IF xRaport THEN
	sDane := '';
	xRaport := FALSE;
	IF intStatus <> intStatusZaraportowana THEN
		intStatusZaraportowana := intStatus;
		fnKomunikatDaneDodaj_xOverFlow(sDane := sDane , sAtrybut := 'STATUS=' , sWartosc := INT_TO_STRING(intStatus) , xOverFlow := xOverFlow);	
		IF xOverFlow = TRUE THEN
			fnZapiszKomunikat(	sCalyKomunikat := '' ,
						sTypKomunikatu := 'M' ,
						sMnemonik := sMnemonik ,
						sMACAdres := sMACAdres ,
						sIDNadawcy := sIdInstancji ,
						sIDOdbiorcy := sIdAplikacji ,
						sDaneZapasowe := sDaneZapasowe ,
						sDane := sDane ,
						arTablicaKomunikatow := arTablicaKomunikatow ,
						intTablicaKomunikatowZnacznikZapisu := intTablicaKomunikatowZnacznikZapisu ,
						intTablicaKomunikatowRozmiar := intTablicaKomunikatowRozmiar ,
						sWyslanyKomunikat := sWyslanyKomunikatDummy);
			sDane := '';
		END_IF	
	END_IF	
	//Napięcia fazowe
	IF rNapiecieL1 <> rNapiecieL1Zaraportowana THEN
		rNapiecieL1Zaraportowana := rNapiecieL1;
		fnKomunikatDaneDodaj_xOverFlow(sDane := sDane , sAtrybut := 'VOLTL1=' , sWartosc := REAL_TO_STRING(rNapiecieL1) , xOverFlow := xOverFlow);	
		IF xOverFlow = TRUE THEN
			fnZapiszKomunikat(	sCalyKomunikat := '' ,
						sTypKomunikatu := 'M' ,
						sMnemonik := sMnemonik ,
						sMACAdres := sMACAdres ,
						sIDNadawcy := sIdInstancji ,
						sIDOdbiorcy := sIdAplikacji ,
						sDaneZapasowe := sDaneZapasowe ,
						sDane := sDane ,
						arTablicaKomunikatow := arTablicaKomunikatow ,
						intTablicaKomunikatowZnacznikZapisu := intTablicaKomunikatowZnacznikZapisu ,
						intTablicaKomunikatowRozmiar := intTablicaKomunikatowRozmiar ,
						sWyslanyKomunikat := sWyslanyKomunikatDummy);
			sDane := '';
		END_IF	
	END_IF
	IF rNapiecieL2 <> rNapiecieL2Zaraportowana THEN
		rNapiecieL2Zaraportowana := rNapiecieL2;
		fnKomunikatDaneDodaj_xOverFlow(sDane := sDane , sAtrybut := 'VOLTL2=' , sWartosc := REAL_TO_STRING(rNapiecieL2) , xOverFlow := xOverFlow);	
		IF xOverFlow = TRUE THEN
			fnZapiszKomunikat(	sCalyKomunikat := '' ,
						sTypKomunikatu := 'M' ,
						sMnemonik := sMnemonik ,
						sMACAdres := sMACAdres ,
						sIDNadawcy := sIdInstancji ,
						sIDOdbiorcy := sIdAplikacji ,
						sDaneZapasowe := sDaneZapasowe ,
						sDane := sDane ,
						arTablicaKomunikatow := arTablicaKomunikatow ,
						intTablicaKomunikatowZnacznikZapisu := intTablicaKomunikatowZnacznikZapisu ,
						intTablicaKomunikatowRozmiar := intTablicaKomunikatowRozmiar ,
						sWyslanyKomunikat := sWyslanyKomunikatDummy);
			sDane := '';
		END_IF	
	END_IF	
	IF rNapiecieL3 <> rNapiecieL3Zaraportowana THEN
		rNapiecieL3Zaraportowana := rNapiecieL3;
		fnKomunikatDaneDodaj_xOverFlow(sDane := sDane , sAtrybut := 'VOLTL3=' , sWartosc := REAL_TO_STRING(rNapiecieL3) , xOverFlow := xOverFlow);
		IF xOverFlow = TRUE THEN
			fnZapiszKomunikat(	sCalyKomunikat := '' ,
						sTypKomunikatu := 'M' ,
						sMnemonik := sMnemonik ,
						sMACAdres := sMACAdres ,
						sIDNadawcy := sIdInstancji ,
						sIDOdbiorcy := sIdAplikacji ,
						sDaneZapasowe := sDaneZapasowe ,
						sDane := sDane ,
						arTablicaKomunikatow := arTablicaKomunikatow ,
						intTablicaKomunikatowZnacznikZapisu := intTablicaKomunikatowZnacznikZapisu ,
						intTablicaKomunikatowRozmiar := intTablicaKomunikatowRozmiar ,
						sWyslanyKomunikat := sWyslanyKomunikatDummy);
			sDane := '';
		END_IF		
	END_IF
	//Napięcia przewodowe		
	IF rNapiecieL1L2 <> rNapiecieL1L2Zaraportowana THEN
		rNapiecieL1L2Zaraportowana := rNapiecieL1L2;
		fnKomunikatDaneDodaj_xOverFlow(sDane := sDane , sAtrybut := 'VOLTL1L2=' , sWartosc := REAL_TO_STRING(rNapiecieL1L2) , xOverFlow := xOverFlow);	
		IF xOverFlow = TRUE THEN
			fnZapiszKomunikat(	sCalyKomunikat := '' ,
						sTypKomunikatu := 'M' ,
						sMnemonik := sMnemonik ,
						sMACAdres := sMACAdres ,
						sIDNadawcy := sIdInstancji ,
						sIDOdbiorcy := sIdAplikacji ,
						sDaneZapasowe := sDaneZapasowe ,
						sDane := sDane ,
						arTablicaKomunikatow := arTablicaKomunikatow ,
						intTablicaKomunikatowZnacznikZapisu := intTablicaKomunikatowZnacznikZapisu ,
						intTablicaKomunikatowRozmiar := intTablicaKomunikatowRozmiar ,
						sWyslanyKomunikat := sWyslanyKomunikatDummy);
			sDane := '';
		END_IF	
	END_IF
	IF rNapiecieL2L3 <> rNapiecieL2L3Zaraportowana THEN
		rNapiecieL2L3Zaraportowana := rNapiecieL2L3;
		fnKomunikatDaneDodaj_xOverFlow(sDane := sDane , sAtrybut := 'VOLTL2L3=' , sWartosc := REAL_TO_STRING(rNapiecieL2L3) , xOverFlow := xOverFlow);	
		IF xOverFlow = TRUE THEN
			fnZapiszKomunikat(	sCalyKomunikat := '' ,
						sTypKomunikatu := 'M' ,
						sMnemonik := sMnemonik ,
						sMACAdres := sMACAdres ,
						sIDNadawcy := sIdInstancji ,
						sIDOdbiorcy := sIdAplikacji ,
						sDaneZapasowe := sDaneZapasowe ,
						sDane := sDane ,
						arTablicaKomunikatow := arTablicaKomunikatow ,
						intTablicaKomunikatowZnacznikZapisu := intTablicaKomunikatowZnacznikZapisu ,
						intTablicaKomunikatowRozmiar := intTablicaKomunikatowRozmiar ,
						sWyslanyKomunikat := sWyslanyKomunikatDummy);
			sDane := '';
		END_IF	
	END_IF	
	IF rNapiecieL3L1 <> rNapiecieL3L1Zaraportowana THEN
		rNapiecieL3L1Zaraportowana := rNapiecieL3L1;
		fnKomunikatDaneDodaj_xOverFlow(sDane := sDane , sAtrybut := 'VOLTL3L1=' , sWartosc := REAL_TO_STRING(rNapiecieL3L1) , xOverFlow := xOverFlow);	
		IF xOverFlow = TRUE THEN
			fnZapiszKomunikat(	sCalyKomunikat := '' ,
						sTypKomunikatu := 'M' ,
						sMnemonik := sMnemonik ,
						sMACAdres := sMACAdres ,
						sIDNadawcy := sIdInstancji ,
						sIDOdbiorcy := sIdAplikacji ,
						sDaneZapasowe := sDaneZapasowe ,
						sDane := sDane ,
						arTablicaKomunikatow := arTablicaKomunikatow ,
						intTablicaKomunikatowZnacznikZapisu := intTablicaKomunikatowZnacznikZapisu ,
						intTablicaKomunikatowRozmiar := intTablicaKomunikatowRozmiar ,
						sWyslanyKomunikat := sWyslanyKomunikatDummy);
			sDane := '';
		END_IF	
	END_IF
	//Częstotliwość 
	IF rCzestotliwosc <> rCzestotliwoscZaraportowana THEN
		rCzestotliwoscZaraportowana := rCzestotliwosc;
		fnKomunikatDaneDodaj_xOverFlow(sDane := sDane , sAtrybut := 'CZEST=' , sWartosc := REAL_TO_STRING(rCzestotliwosc) , xOverFlow := xOverFlow);	
		IF xOverFlow = TRUE THEN
			fnZapiszKomunikat(	sCalyKomunikat := '' ,
						sTypKomunikatu := 'M' ,
						sMnemonik := sMnemonik ,
						sMACAdres := sMACAdres ,
						sIDNadawcy := sIdInstancji ,
						sIDOdbiorcy := sIdAplikacji ,
						sDaneZapasowe := sDaneZapasowe ,
						sDane := sDane ,
						arTablicaKomunikatow := arTablicaKomunikatow ,
						intTablicaKomunikatowZnacznikZapisu := intTablicaKomunikatowZnacznikZapisu ,
						intTablicaKomunikatowRozmiar := intTablicaKomunikatowRozmiar ,
						sWyslanyKomunikat := sWyslanyKomunikatDummy);
			sDane := '';
		END_IF	
	END_IF
	//Czas pracy 
	IF rCzasPracyAnalizatora <> rCzasPracyAnalizatoraZaraportowana THEN
		rCzasPracyAnalizatoraZaraportowana := rCzasPracyAnalizatora;
		fnKomunikatDaneDodaj_xOverFlow(sDane := sDane , sAtrybut := 'CZAS=' , sWartosc := REAL_TO_STRING(rCzasPracyAnalizatora) , xOverFlow := xOverFlow);	
		IF xOverFlow = TRUE THEN
			fnZapiszKomunikat(	sCalyKomunikat := '' ,
						sTypKomunikatu := 'M' ,
						sMnemonik := sMnemonik ,
						sMACAdres := sMACAdres ,
						sIDNadawcy := sIdInstancji ,
						sIDOdbiorcy := sIdAplikacji ,
						sDaneZapasowe := sDaneZapasowe ,
						sDane := sDane ,
						arTablicaKomunikatow := arTablicaKomunikatow ,
						intTablicaKomunikatowZnacznikZapisu := intTablicaKomunikatowZnacznikZapisu ,
						intTablicaKomunikatowRozmiar := intTablicaKomunikatowRozmiar ,
						sWyslanyKomunikat := sWyslanyKomunikatDummy);
			sDane := '';
		END_IF	
	END_IF
	//Prądy fazowe	
	IF rPradL1 <> rPradL1Zaraportowana THEN
		rPradL1Zaraportowana := rPradL1;
		fnKomunikatDaneDodaj_xOverFlow(sDane := sDane , sAtrybut := 'AMPERL1=' , sWartosc := REAL_TO_STRING(rPradL1) , xOverFlow := xOverFlow);	
		IF xOverFlow = TRUE THEN
			fnZapiszKomunikat(	sCalyKomunikat := '' ,
						sTypKomunikatu := 'M' ,
						sMnemonik := sMnemonik ,
						sMACAdres := sMACAdres ,
						sIDNadawcy := sIdInstancji ,
						sIDOdbiorcy := sIdAplikacji ,
						sDaneZapasowe := sDaneZapasowe ,
						sDane := sDane ,
						arTablicaKomunikatow := arTablicaKomunikatow ,
						intTablicaKomunikatowZnacznikZapisu := intTablicaKomunikatowZnacznikZapisu ,
						intTablicaKomunikatowRozmiar := intTablicaKomunikatowRozmiar ,
						sWyslanyKomunikat := sWyslanyKomunikatDummy);
			sDane := '';
		END_IF	
	END_IF
	IF rPradL2 <> rPradL2Zaraportowana THEN
		rPradL2Zaraportowana := rPradL2;
		fnKomunikatDaneDodaj_xOverFlow(sDane := sDane , sAtrybut := 'AMPERL2=' , sWartosc := REAL_TO_STRING(rPradL2) , xOverFlow := xOverFlow);	
		IF xOverFlow = TRUE THEN
			fnZapiszKomunikat(	sCalyKomunikat := '' ,
						sTypKomunikatu := 'M' ,
						sMnemonik := sMnemonik ,
						sMACAdres := sMACAdres ,
						sIDNadawcy := sIdInstancji ,
						sIDOdbiorcy := sIdAplikacji ,
						sDaneZapasowe := sDaneZapasowe ,
						sDane := sDane ,
						arTablicaKomunikatow := arTablicaKomunikatow ,
						intTablicaKomunikatowZnacznikZapisu := intTablicaKomunikatowZnacznikZapisu ,
						intTablicaKomunikatowRozmiar := intTablicaKomunikatowRozmiar ,
						sWyslanyKomunikat := sWyslanyKomunikatDummy);
			sDane := '';
		END_IF	
	END_IF	
	IF rPradL3 <> rPradL3Zaraportowana THEN
		rPradL3Zaraportowana := rPradL3;
		fnKomunikatDaneDodaj_xOverFlow(sDane := sDane , sAtrybut := 'AMPERL3=' , sWartosc := REAL_TO_STRING(rPradL3) , xOverFlow := xOverFlow);	
		IF xOverFlow = TRUE THEN
			fnZapiszKomunikat(	sCalyKomunikat := '' ,
						sTypKomunikatu := 'M' ,
						sMnemonik := sMnemonik ,
						sMACAdres := sMACAdres ,
						sIDNadawcy := sIdInstancji ,
						sIDOdbiorcy := sIdAplikacji ,
						sDaneZapasowe := sDaneZapasowe ,
						sDane := sDane ,
						arTablicaKomunikatow := arTablicaKomunikatow ,
						intTablicaKomunikatowZnacznikZapisu := intTablicaKomunikatowZnacznikZapisu ,
						intTablicaKomunikatowRozmiar := intTablicaKomunikatowRozmiar ,
						sWyslanyKomunikat := sWyslanyKomunikatDummy);
			sDane := '';
		END_IF	
	END_IF
	IF rPradN <> rPradNZaraportowana THEN
		rPradNZaraportowana := rPradN;
		fnKomunikatDaneDodaj_xOverFlow(sDane := sDane , sAtrybut := 'AMPERN=' , sWartosc := REAL_TO_STRING(rPradN) , xOverFlow := xOverFlow);	
		IF xOverFlow = TRUE THEN
			fnZapiszKomunikat(	sCalyKomunikat := '' ,
						sTypKomunikatu := 'M' ,
						sMnemonik := sMnemonik ,
						sMACAdres := sMACAdres ,
						sIDNadawcy := sIdInstancji ,
						sIDOdbiorcy := sIdAplikacji ,
						sDaneZapasowe := sDaneZapasowe ,
						sDane := sDane ,
						arTablicaKomunikatow := arTablicaKomunikatow ,
						intTablicaKomunikatowZnacznikZapisu := intTablicaKomunikatowZnacznikZapisu ,
						intTablicaKomunikatowRozmiar := intTablicaKomunikatowRozmiar ,
						sWyslanyKomunikat := sWyslanyKomunikatDummy);
			sDane := '';
		END_IF	
	END_IF
	//Prądy średnie fazowe
	IF rPradSredniL1 <> rPradSredniL1Zaraportowana THEN
		rPradSredniL1Zaraportowana := rPradSredniL1;
		fnKomunikatDaneDodaj_xOverFlow(sDane := sDane , sAtrybut := 'AMPERAVGL1=' , sWartosc := REAL_TO_STRING(rPradSredniL1) , xOverFlow := xOverFlow);	
		IF xOverFlow = TRUE THEN
			fnZapiszKomunikat(	sCalyKomunikat := '' ,
						sTypKomunikatu := 'M' ,
						sMnemonik := sMnemonik ,
						sMACAdres := sMACAdres ,
						sIDNadawcy := sIdInstancji ,
						sIDOdbiorcy := sIdAplikacji ,
						sDaneZapasowe := sDaneZapasowe ,
						sDane := sDane ,
						arTablicaKomunikatow := arTablicaKomunikatow ,
						intTablicaKomunikatowZnacznikZapisu := intTablicaKomunikatowZnacznikZapisu ,
						intTablicaKomunikatowRozmiar := intTablicaKomunikatowRozmiar ,
						sWyslanyKomunikat := sWyslanyKomunikatDummy);
			sDane := '';
		END_IF	
	END_IF
	IF rPradSredniL2 <> rPradSredniL2Zaraportowana THEN
		rPradSredniL2Zaraportowana := rPradSredniL2;
		fnKomunikatDaneDodaj_xOverFlow(sDane := sDane , sAtrybut := 'AMPERAVGL2=' , sWartosc := REAL_TO_STRING(rPradSredniL2) , xOverFlow := xOverFlow);	
		IF xOverFlow = TRUE THEN
			fnZapiszKomunikat(	sCalyKomunikat := '' ,
						sTypKomunikatu := 'M' ,
						sMnemonik := sMnemonik ,
						sMACAdres := sMACAdres ,
						sIDNadawcy := sIdInstancji ,
						sIDOdbiorcy := sIdAplikacji ,
						sDaneZapasowe := sDaneZapasowe ,
						sDane := sDane ,
						arTablicaKomunikatow := arTablicaKomunikatow ,
						intTablicaKomunikatowZnacznikZapisu := intTablicaKomunikatowZnacznikZapisu ,
						intTablicaKomunikatowRozmiar := intTablicaKomunikatowRozmiar ,
						sWyslanyKomunikat := sWyslanyKomunikatDummy);
			sDane := '';
		END_IF	
	END_IF	
	IF rPradSredniL3 <> rPradSredniL3Zaraportowana THEN
		rPradSredniL3Zaraportowana := rPradSredniL3;
		fnKomunikatDaneDodaj_xOverFlow(sDane := sDane , sAtrybut := 'AMPERAVGL3=' , sWartosc := REAL_TO_STRING(rPradSredniL3) , xOverFlow := xOverFlow);
		IF xOverFlow = TRUE THEN
			fnZapiszKomunikat(	sCalyKomunikat := '' ,
						sTypKomunikatu := 'M' ,
						sMnemonik := sMnemonik ,
						sMACAdres := sMACAdres ,
						sIDNadawcy := sIdInstancji ,
						sIDOdbiorcy := sIdAplikacji ,
						sDaneZapasowe := sDaneZapasowe ,
						sDane := sDane ,
						arTablicaKomunikatow := arTablicaKomunikatow ,
						intTablicaKomunikatowZnacznikZapisu := intTablicaKomunikatowZnacznikZapisu ,
						intTablicaKomunikatowRozmiar := intTablicaKomunikatowRozmiar ,
						sWyslanyKomunikat := sWyslanyKomunikatDummy);
			sDane := '';
		END_IF	
	END_IF
	//Prąd średni
	IF rPradSredni <> rPradSredniZaraportowana THEN
		rPradSredniZaraportowana := rPradSredni;
		fnKomunikatDaneDodaj_xOverFlow(sDane := sDane , sAtrybut := 'AMPERAVG=' , sWartosc := REAL_TO_STRING(rPradSredni) , xOverFlow := xOverFlow);
		IF xOverFlow = TRUE THEN
			fnZapiszKomunikat(	sCalyKomunikat := '' ,
						sTypKomunikatu := 'M' ,
						sMnemonik := sMnemonik ,
						sMACAdres := sMACAdres ,
						sIDNadawcy := sIdInstancji ,
						sIDOdbiorcy := sIdAplikacji ,
						sDaneZapasowe := sDaneZapasowe ,
						sDane := sDane ,
						arTablicaKomunikatow := arTablicaKomunikatow ,
						intTablicaKomunikatowZnacznikZapisu := intTablicaKomunikatowZnacznikZapisu ,
						intTablicaKomunikatowRozmiar := intTablicaKomunikatowRozmiar ,
						sWyslanyKomunikat := sWyslanyKomunikatDummy);
			sDane := '';
		END_IF	
	END_IF
	//Moce 3-fazowe		 
	IF rMocCzynnaCalkowita <> rMocCzynnaCalkowitaZaraportowana THEN
		rMocCzynnaCalkowitaZaraportowana := rMocCzynnaCalkowita;
		fnKomunikatDaneDodaj_xOverFlow(sDane := sDane , sAtrybut := 'POWCE=' , sWartosc := REAL_TO_STRING(rMocCzynnaCalkowita) , xOverFlow := xOverFlow);
		IF xOverFlow = TRUE THEN
			fnZapiszKomunikat(	sCalyKomunikat := '' ,
						sTypKomunikatu := 'M' ,
						sMnemonik := sMnemonik ,
						sMACAdres := sMACAdres ,
						sIDNadawcy := sIdInstancji ,
						sIDOdbiorcy := sIdAplikacji ,
						sDaneZapasowe := sDaneZapasowe ,
						sDane := sDane ,
						arTablicaKomunikatow := arTablicaKomunikatow ,
						intTablicaKomunikatowZnacznikZapisu := intTablicaKomunikatowZnacznikZapisu ,
						intTablicaKomunikatowRozmiar := intTablicaKomunikatowRozmiar ,
						sWyslanyKomunikat := sWyslanyKomunikatDummy);
			sDane := '';
		END_IF	
	END_IF
	IF rMocBiernaCalkowita <> rMocBiernaCalkowitaZaraportowana THEN
		rMocBiernaCalkowitaZaraportowana := rMocBiernaCalkowita;
		fnKomunikatDaneDodaj_xOverFlow(sDane := sDane , sAtrybut := 'POWBE=' , sWartosc := REAL_TO_STRING(rMocBiernaCalkowita) , xOverFlow := xOverFlow);	
		IF xOverFlow = TRUE THEN
			fnZapiszKomunikat(	sCalyKomunikat := '' ,
						sTypKomunikatu := 'M' ,
						sMnemonik := sMnemonik ,
						sMACAdres := sMACAdres ,
						sIDNadawcy := sIdInstancji ,
						sIDOdbiorcy := sIdAplikacji ,
						sDaneZapasowe := sDaneZapasowe ,
						sDane := sDane ,
						arTablicaKomunikatow := arTablicaKomunikatow ,
						intTablicaKomunikatowZnacznikZapisu := intTablicaKomunikatowZnacznikZapisu ,
						intTablicaKomunikatowRozmiar := intTablicaKomunikatowRozmiar ,
						sWyslanyKomunikat := sWyslanyKomunikatDummy);
			sDane := '';
		END_IF	
	END_IF	
	IF rMocPozornaCalkowita <> rMocPozornaCalkowitaZaraportowana THEN
		rMocPozornaCalkowitaZaraportowana := rMocPozornaCalkowita;
		fnKomunikatDaneDodaj_xOverFlow(sDane := sDane , sAtrybut := 'POWPE=' , sWartosc := REAL_TO_STRING(rMocPozornaCalkowita) , xOverFlow := xOverFlow);	
		IF xOverFlow = TRUE THEN
			fnZapiszKomunikat(	sCalyKomunikat := '' ,
						sTypKomunikatu := 'M' ,
						sMnemonik := sMnemonik ,
						sMACAdres := sMACAdres ,
						sIDNadawcy := sIdInstancji ,
						sIDOdbiorcy := sIdAplikacji ,
						sDaneZapasowe := sDaneZapasowe ,
						sDane := sDane ,
						arTablicaKomunikatow := arTablicaKomunikatow ,
						intTablicaKomunikatowZnacznikZapisu := intTablicaKomunikatowZnacznikZapisu ,
						intTablicaKomunikatowRozmiar := intTablicaKomunikatowRozmiar ,
						sWyslanyKomunikat := sWyslanyKomunikatDummy);
			sDane := '';
		END_IF	
	END_IF
	//Współczynnik mocy 3-fazowy
	IF rWspolczynnikMocyCalkowity <> rWspolczynnikMocyCalkowityZaraportowana THEN
		rWspolczynnikMocyCalkowityZaraportowana := rWspolczynnikMocyCalkowity;
		fnKomunikatDaneDodaj_xOverFlow(sDane := sDane , sAtrybut := 'FACTOR3PH=' , sWartosc := REAL_TO_STRING(rWspolczynnikMocyCalkowity) , xOverFlow := xOverFlow);	
		IF xOverFlow = TRUE THEN
			fnZapiszKomunikat(	sCalyKomunikat := '' ,
						sTypKomunikatu := 'M' ,
						sMnemonik := sMnemonik ,
						sMACAdres := sMACAdres ,
						sIDNadawcy := sIdInstancji ,
						sIDOdbiorcy := sIdAplikacji ,
						sDaneZapasowe := sDaneZapasowe ,
						sDane := sDane ,
						arTablicaKomunikatow := arTablicaKomunikatow ,
						intTablicaKomunikatowZnacznikZapisu := intTablicaKomunikatowZnacznikZapisu ,
						intTablicaKomunikatowRozmiar := intTablicaKomunikatowRozmiar ,
						sWyslanyKomunikat := sWyslanyKomunikatDummy);
			sDane := '';
		END_IF	
	END_IF
	//Moce czynne fazowe
	IF rMocCzynnaL1 <> rMocCzynnaL1Zaraportowana THEN
		rMocCzynnaL1Zaraportowana := rMocCzynnaL1;
		fnKomunikatDaneDodaj_xOverFlow(sDane := sDane , sAtrybut := 'POWCECL1=' , sWartosc := REAL_TO_STRING(rMocCzynnaL1) , xOverFlow := xOverFlow);	
		IF xOverFlow = TRUE THEN
			fnZapiszKomunikat(	sCalyKomunikat := '' ,
						sTypKomunikatu := 'M' ,
						sMnemonik := sMnemonik ,
						sMACAdres := sMACAdres ,
						sIDNadawcy := sIdInstancji ,
						sIDOdbiorcy := sIdAplikacji ,
						sDaneZapasowe := sDaneZapasowe ,
						sDane := sDane ,
						arTablicaKomunikatow := arTablicaKomunikatow ,
						intTablicaKomunikatowZnacznikZapisu := intTablicaKomunikatowZnacznikZapisu ,
						intTablicaKomunikatowRozmiar := intTablicaKomunikatowRozmiar ,
						sWyslanyKomunikat := sWyslanyKomunikatDummy);
			sDane := '';
		END_IF	
	END_IF
	IF rMocCzynnaL2 <> rMocCzynnaL2Zaraportowana THEN
		rMocCzynnaL2Zaraportowana := rMocCzynnaL2;
		fnKomunikatDaneDodaj_xOverFlow(sDane := sDane , sAtrybut := 'POWCECL2=' , sWartosc := REAL_TO_STRING(rMocCzynnaL2) , xOverFlow := xOverFlow);	
		IF xOverFlow = TRUE THEN
			fnZapiszKomunikat(	sCalyKomunikat := '' ,
						sTypKomunikatu := 'M' ,
						sMnemonik := sMnemonik ,
						sMACAdres := sMACAdres ,
						sIDNadawcy := sIdInstancji ,
						sIDOdbiorcy := sIdAplikacji ,
						sDaneZapasowe := sDaneZapasowe ,
						sDane := sDane ,
						arTablicaKomunikatow := arTablicaKomunikatow ,
						intTablicaKomunikatowZnacznikZapisu := intTablicaKomunikatowZnacznikZapisu ,
						intTablicaKomunikatowRozmiar := intTablicaKomunikatowRozmiar ,
						sWyslanyKomunikat := sWyslanyKomunikatDummy);
			sDane := '';
		END_IF	
	END_IF
	IF rMocCzynnaL3 <> rMocCzynnaL3Zaraportowana THEN
		rMocCzynnaL3Zaraportowana := rMocCzynnaL3;
		fnKomunikatDaneDodaj_xOverFlow(sDane := sDane , sAtrybut := 'POWCECL3=' , sWartosc := REAL_TO_STRING(rMocCzynnaL3) , xOverFlow := xOverFlow);
		IF xOverFlow = TRUE THEN
			fnZapiszKomunikat(	sCalyKomunikat := '' ,
						sTypKomunikatu := 'M' ,
						sMnemonik := sMnemonik ,
						sMACAdres := sMACAdres ,
						sIDNadawcy := sIdInstancji ,
						sIDOdbiorcy := sIdAplikacji ,
						sDaneZapasowe := sDaneZapasowe ,
						sDane := sDane ,
						arTablicaKomunikatow := arTablicaKomunikatow ,
						intTablicaKomunikatowZnacznikZapisu := intTablicaKomunikatowZnacznikZapisu ,
						intTablicaKomunikatowRozmiar := intTablicaKomunikatowRozmiar ,
						sWyslanyKomunikat := sWyslanyKomunikatDummy);
			sDane := '';
		END_IF		
	END_IF
	//Moce bierne fazowe	
	IF rMocBiernaL1 <> rMocBiernaL1Zaraportowana THEN
		rMocBiernaL1Zaraportowana := rMocBiernaL1;
		fnKomunikatDaneDodaj_xOverFlow(sDane := sDane , sAtrybut := 'POWCEBL1=' , sWartosc := REAL_TO_STRING(rMocBiernaL1) , xOverFlow := xOverFlow);	
		IF xOverFlow = TRUE THEN
			fnZapiszKomunikat(	sCalyKomunikat := '' ,
						sTypKomunikatu := 'M' ,
						sMnemonik := sMnemonik ,
						sMACAdres := sMACAdres ,
						sIDNadawcy := sIdInstancji ,
						sIDOdbiorcy := sIdAplikacji ,
						sDaneZapasowe := sDaneZapasowe ,
						sDane := sDane ,
						arTablicaKomunikatow := arTablicaKomunikatow ,
						intTablicaKomunikatowZnacznikZapisu := intTablicaKomunikatowZnacznikZapisu ,
						intTablicaKomunikatowRozmiar := intTablicaKomunikatowRozmiar ,
						sWyslanyKomunikat := sWyslanyKomunikatDummy);
			sDane := '';
		END_IF	
	END_IF
	IF rMocBiernaL2 <> rMocBiernaL2Zaraportowana THEN
		rMocBiernaL2Zaraportowana := rMocBiernaL2;
		fnKomunikatDaneDodaj_xOverFlow(sDane := sDane , sAtrybut := 'POWCEBL2=' , sWartosc := REAL_TO_STRING(rMocBiernaL2) , xOverFlow := xOverFlow);	
		IF xOverFlow = TRUE THEN
			fnZapiszKomunikat(	sCalyKomunikat := '' ,
						sTypKomunikatu := 'M' ,
						sMnemonik := sMnemonik ,
						sMACAdres := sMACAdres ,
						sIDNadawcy := sIdInstancji ,
						sIDOdbiorcy := sIdAplikacji ,
						sDaneZapasowe := sDaneZapasowe ,
						sDane := sDane ,
						arTablicaKomunikatow := arTablicaKomunikatow ,
						intTablicaKomunikatowZnacznikZapisu := intTablicaKomunikatowZnacznikZapisu ,
						intTablicaKomunikatowRozmiar := intTablicaKomunikatowRozmiar ,
						sWyslanyKomunikat := sWyslanyKomunikatDummy);
			sDane := '';
		END_IF	
	END_IF
	IF rMocBiernaL3 <> rMocBiernaL3Zaraportowana THEN
		rMocBiernaL3Zaraportowana := rMocBiernaL3;
		fnKomunikatDaneDodaj_xOverFlow(sDane := sDane , sAtrybut := 'POWCEBL3=' , sWartosc := REAL_TO_STRING(rMocBiernaL3) , xOverFlow := xOverFlow);	
		IF xOverFlow = TRUE THEN
			fnZapiszKomunikat(	sCalyKomunikat := '' ,
						sTypKomunikatu := 'M' ,
						sMnemonik := sMnemonik ,
						sMACAdres := sMACAdres ,
						sIDNadawcy := sIdInstancji ,
						sIDOdbiorcy := sIdAplikacji ,
						sDaneZapasowe := sDaneZapasowe ,
						sDane := sDane ,
						arTablicaKomunikatow := arTablicaKomunikatow ,
						intTablicaKomunikatowZnacznikZapisu := intTablicaKomunikatowZnacznikZapisu ,
						intTablicaKomunikatowRozmiar := intTablicaKomunikatowRozmiar ,
						sWyslanyKomunikat := sWyslanyKomunikatDummy);
			sDane := '';
		END_IF	
	END_IF
	//Moce pozorne fazowe
	IF rMocPozornaL1 <> rMocPozornaL1Zaraportowana THEN
		rMocPozornaL1Zaraportowana := rMocPozornaL1;
		fnKomunikatDaneDodaj_xOverFlow(sDane := sDane , sAtrybut := 'POWCEPL1=' , sWartosc := REAL_TO_STRING(rMocPozornaL1) , xOverFlow := xOverFlow);	
		IF xOverFlow = TRUE THEN
			fnZapiszKomunikat(	sCalyKomunikat := '' ,
						sTypKomunikatu := 'M' ,
						sMnemonik := sMnemonik ,
						sMACAdres := sMACAdres ,
						sIDNadawcy := sIdInstancji ,
						sIDOdbiorcy := sIdAplikacji ,
						sDaneZapasowe := sDaneZapasowe ,
						sDane := sDane ,
						arTablicaKomunikatow := arTablicaKomunikatow ,
						intTablicaKomunikatowZnacznikZapisu := intTablicaKomunikatowZnacznikZapisu ,
						intTablicaKomunikatowRozmiar := intTablicaKomunikatowRozmiar ,
						sWyslanyKomunikat := sWyslanyKomunikatDummy);
			sDane := '';
		END_IF	
	END_IF
	IF rMocPozornaL2 <> rMocPozornaL2Zaraportowana THEN
		rMocPozornaL2Zaraportowana := rMocPozornaL2;
		fnKomunikatDaneDodaj_xOverFlow(sDane := sDane , sAtrybut := 'POWCEPL2=' , sWartosc := REAL_TO_STRING(rMocPozornaL2) , xOverFlow := xOverFlow);	
		IF xOverFlow = TRUE THEN
			fnZapiszKomunikat(	sCalyKomunikat := '' ,
						sTypKomunikatu := 'M' ,
						sMnemonik := sMnemonik ,
						sMACAdres := sMACAdres ,
						sIDNadawcy := sIdInstancji ,
						sIDOdbiorcy := sIdAplikacji ,
						sDaneZapasowe := sDaneZapasowe ,
						sDane := sDane ,
						arTablicaKomunikatow := arTablicaKomunikatow ,
						intTablicaKomunikatowZnacznikZapisu := intTablicaKomunikatowZnacznikZapisu ,
						intTablicaKomunikatowRozmiar := intTablicaKomunikatowRozmiar ,
						sWyslanyKomunikat := sWyslanyKomunikatDummy);
			sDane := '';
		END_IF	
	END_IF
	IF rMocPozornaL3 <> rMocPozornaL3Zaraportowana THEN
		rMocPozornaL3Zaraportowana := rMocPozornaL3;
		fnKomunikatDaneDodaj_xOverFlow(sDane := sDane , sAtrybut := 'POWCEPL3=' , sWartosc := REAL_TO_STRING(rMocPozornaL3) , xOverFlow := xOverFlow);	
		IF xOverFlow = TRUE THEN
			fnZapiszKomunikat(	sCalyKomunikat := '' ,
						sTypKomunikatu := 'M' ,
						sMnemonik := sMnemonik ,
						sMACAdres := sMACAdres ,
						sIDNadawcy := sIdInstancji ,
						sIDOdbiorcy := sIdAplikacji ,
						sDaneZapasowe := sDaneZapasowe ,
						sDane := sDane ,
						arTablicaKomunikatow := arTablicaKomunikatow ,
						intTablicaKomunikatowZnacznikZapisu := intTablicaKomunikatowZnacznikZapisu ,
						intTablicaKomunikatowRozmiar := intTablicaKomunikatowRozmiar ,
						sWyslanyKomunikat := sWyslanyKomunikatDummy);
			sDane := '';
		END_IF	
	END_IF
	//Współczynniki mocy fazowe
	IF rWspolczynnikMocyL1 <> rWspolczynnikMocyL1Zaraportowana THEN
		rWspolczynnikMocyL1Zaraportowana := rWspolczynnikMocyL1;
		fnKomunikatDaneDodaj_xOverFlow(sDane := sDane , sAtrybut := 'FACTORL1=' , sWartosc := REAL_TO_STRING(rWspolczynnikMocyL1) , xOverFlow := xOverFlow);
		IF xOverFlow = TRUE THEN
			fnZapiszKomunikat(	sCalyKomunikat := '' ,
						sTypKomunikatu := 'M' ,
						sMnemonik := sMnemonik ,
						sMACAdres := sMACAdres ,
						sIDNadawcy := sIdInstancji ,
						sIDOdbiorcy := sIdAplikacji ,
						sDaneZapasowe := sDaneZapasowe ,
						sDane := sDane ,
						arTablicaKomunikatow := arTablicaKomunikatow ,
						intTablicaKomunikatowZnacznikZapisu := intTablicaKomunikatowZnacznikZapisu ,
						intTablicaKomunikatowRozmiar := intTablicaKomunikatowRozmiar ,
						sWyslanyKomunikat := sWyslanyKomunikatDummy);
			sDane := '';
		END_IF		
	END_IF
	IF rWspolczynnikMocyL2 <> rWspolczynnikMocyL2Zaraportowana THEN
		rWspolczynnikMocyL2Zaraportowana := rWspolczynnikMocyL2;
		fnKomunikatDaneDodaj_xOverFlow(sDane := sDane , sAtrybut := 'FACTORL2=' , sWartosc := REAL_TO_STRING(rWspolczynnikMocyL2) , xOverFlow := xOverFlow);	
		IF xOverFlow = TRUE THEN
			fnZapiszKomunikat(	sCalyKomunikat := '' ,
						sTypKomunikatu := 'M' ,
						sMnemonik := sMnemonik ,
						sMACAdres := sMACAdres ,
						sIDNadawcy := sIdInstancji ,
						sIDOdbiorcy := sIdAplikacji ,
						sDaneZapasowe := sDaneZapasowe ,
						sDane := sDane ,
						arTablicaKomunikatow := arTablicaKomunikatow ,
						intTablicaKomunikatowZnacznikZapisu := intTablicaKomunikatowZnacznikZapisu ,
						intTablicaKomunikatowRozmiar := intTablicaKomunikatowRozmiar ,
						sWyslanyKomunikat := sWyslanyKomunikatDummy);
			sDane := '';
		END_IF	
	END_IF
	IF rWspolczynnikMocyL3 <> rWspolczynnikMocyL3Zaraportowana THEN
		rWspolczynnikMocyL3Zaraportowana := rWspolczynnikMocyL3;
		fnKomunikatDaneDodaj_xOverFlow(sDane := sDane , sAtrybut := 'FACTORL3=' , sWartosc := REAL_TO_STRING(rWspolczynnikMocyL3) , xOverFlow := xOverFlow);	
		IF xOverFlow = TRUE THEN
			fnZapiszKomunikat(	sCalyKomunikat := '' ,
						sTypKomunikatu := 'M' ,
						sMnemonik := sMnemonik ,
						sMACAdres := sMACAdres ,
						sIDNadawcy := sIdInstancji ,
						sIDOdbiorcy := sIdAplikacji ,
						sDaneZapasowe := sDaneZapasowe ,
						sDane := sDane ,
						arTablicaKomunikatow := arTablicaKomunikatow ,
						intTablicaKomunikatowZnacznikZapisu := intTablicaKomunikatowZnacznikZapisu ,
						intTablicaKomunikatowRozmiar := intTablicaKomunikatowRozmiar ,
						sWyslanyKomunikat := sWyslanyKomunikatDummy);
			sDane := '';
		END_IF	
	END_IF
	//Energia pobrana
	IF rEnergiaCzynnaPobrana <> rEnergiaCzynnaPobranaZaraportowana THEN
		rEnergiaCzynnaPobranaZaraportowana := rEnergiaCzynnaPobrana;
		fnKomunikatDaneDodaj_xOverFlow(sDane := sDane , sAtrybut := 'ENCE=' , sWartosc := REAL_TO_STRING(rEnergiaCzynnaPobrana) , xOverFlow := xOverFlow);	
		IF xOverFlow = TRUE THEN
			fnZapiszKomunikat(	sCalyKomunikat := '' ,
						sTypKomunikatu := 'M' ,
						sMnemonik := sMnemonik ,
						sMACAdres := sMACAdres ,
						sIDNadawcy := sIdInstancji ,
						sIDOdbiorcy := sIdAplikacji ,
						sDaneZapasowe := sDaneZapasowe ,
						sDane := sDane ,
						arTablicaKomunikatow := arTablicaKomunikatow ,
						intTablicaKomunikatowZnacznikZapisu := intTablicaKomunikatowZnacznikZapisu ,
						intTablicaKomunikatowRozmiar := intTablicaKomunikatowRozmiar ,
						sWyslanyKomunikat := sWyslanyKomunikatDummy);
			sDane := '';
		END_IF	
	END_IF
	IF rEnergiaBiernaPobrana <> rEnergiaBiernaPobranaZaraportowana THEN
		rEnergiaBiernaPobranaZaraportowana := rEnergiaBiernaPobrana;
		fnKomunikatDaneDodaj_xOverFlow(sDane := sDane , sAtrybut := 'ENBE=' , sWartosc := REAL_TO_STRING(rEnergiaBiernaPobrana) , xOverFlow := xOverFlow);	
		IF xOverFlow = TRUE THEN
			fnZapiszKomunikat(	sCalyKomunikat := '' ,
						sTypKomunikatu := 'M' ,
						sMnemonik := sMnemonik ,
						sMACAdres := sMACAdres ,
						sIDNadawcy := sIdInstancji ,
						sIDOdbiorcy := sIdAplikacji ,
						sDaneZapasowe := sDaneZapasowe ,
						sDane := sDane ,
						arTablicaKomunikatow := arTablicaKomunikatow ,
						intTablicaKomunikatowZnacznikZapisu := intTablicaKomunikatowZnacznikZapisu ,
						intTablicaKomunikatowRozmiar := intTablicaKomunikatowRozmiar ,
						sWyslanyKomunikat := sWyslanyKomunikatDummy);
			sDane := '';
		END_IF	
	END_IF
	IF rEnergiaPozornaPobrana <> rEnergiaPozornaPobranaZaraportowana THEN
		rEnergiaPozornaPobranaZaraportowana := rEnergiaPozornaPobrana;
		fnKomunikatDaneDodaj_xOverFlow(sDane := sDane , sAtrybut := 'ENPE=' , sWartosc := REAL_TO_STRING(rEnergiaPozornaPobrana) , xOverFlow := xOverFlow);	
		IF xOverFlow = TRUE THEN
			fnZapiszKomunikat(	sCalyKomunikat := '' ,
						sTypKomunikatu := 'M' ,
						sMnemonik := sMnemonik ,
						sMACAdres := sMACAdres ,
						sIDNadawcy := sIdInstancji ,
						sIDOdbiorcy := sIdAplikacji ,
						sDaneZapasowe := sDaneZapasowe ,
						sDane := sDane ,
						arTablicaKomunikatow := arTablicaKomunikatow ,
						intTablicaKomunikatowZnacznikZapisu := intTablicaKomunikatowZnacznikZapisu ,
						intTablicaKomunikatowRozmiar := intTablicaKomunikatowRozmiar ,
						sWyslanyKomunikat := sWyslanyKomunikatDummy);
			sDane := '';
		END_IF	
	END_IF
	//Moce średnie	
	IF rMocCzynnaSrednia <> rMocCzynnaSredniaZaraportowana THEN
		rMocCzynnaSredniaZaraportowana := rMocCzynnaSrednia;
		fnKomunikatDaneDodaj_xOverFlow(sDane := sDane , sAtrybut := 'POWAVGEC=' , sWartosc := REAL_TO_STRING(rMocCzynnaSrednia) , xOverFlow := xOverFlow);	
		IF xOverFlow = TRUE THEN
			fnZapiszKomunikat(	sCalyKomunikat := '' ,
						sTypKomunikatu := 'M' ,
						sMnemonik := sMnemonik ,
						sMACAdres := sMACAdres ,
						sIDNadawcy := sIdInstancji ,
						sIDOdbiorcy := sIdAplikacji ,
						sDaneZapasowe := sDaneZapasowe ,
						sDane := sDane ,
						arTablicaKomunikatow := arTablicaKomunikatow ,
						intTablicaKomunikatowZnacznikZapisu := intTablicaKomunikatowZnacznikZapisu ,
						intTablicaKomunikatowRozmiar := intTablicaKomunikatowRozmiar ,
						sWyslanyKomunikat := sWyslanyKomunikatDummy);
			sDane := '';
		END_IF	
	END_IF
	IF rMocBiernaSrednia <> rMocBiernaSredniaZaraportowana THEN
		rMocBiernaSredniaZaraportowana := rMocBiernaSrednia;
		fnKomunikatDaneDodaj_xOverFlow(sDane := sDane , sAtrybut := 'POWAVGEB=' , sWartosc := REAL_TO_STRING(rMocBiernaSrednia) , xOverFlow := xOverFlow);	
		IF xOverFlow = TRUE THEN
			fnZapiszKomunikat(	sCalyKomunikat := '' ,
						sTypKomunikatu := 'M' ,
						sMnemonik := sMnemonik ,
						sMACAdres := sMACAdres ,
						sIDNadawcy := sIdInstancji ,
						sIDOdbiorcy := sIdAplikacji ,
						sDaneZapasowe := sDaneZapasowe ,
						sDane := sDane ,
						arTablicaKomunikatow := arTablicaKomunikatow ,
						intTablicaKomunikatowZnacznikZapisu := intTablicaKomunikatowZnacznikZapisu ,
						intTablicaKomunikatowRozmiar := intTablicaKomunikatowRozmiar ,
						sWyslanyKomunikat := sWyslanyKomunikatDummy);
			sDane := '';
		END_IF	
	END_IF
	IF rMocPozornaSrednia <> rMocPozornaSredniaZaraportowana THEN
		rMocPozornaSredniaZaraportowana := rMocPozornaSrednia;
		fnKomunikatDaneDodaj_xOverFlow(sDane := sDane , sAtrybut := 'POWAVGEP=' , sWartosc := REAL_TO_STRING(rMocPozornaSrednia) , xOverFlow := xOverFlow);	
		IF xOverFlow = TRUE THEN
			fnZapiszKomunikat(	sCalyKomunikat := '' ,
						sTypKomunikatu := 'M' ,
						sMnemonik := sMnemonik ,
						sMACAdres := sMACAdres ,
						sIDNadawcy := sIdInstancji ,
						sIDOdbiorcy := sIdAplikacji ,
						sDaneZapasowe := sDaneZapasowe ,
						sDane := sDane ,
						arTablicaKomunikatow := arTablicaKomunikatow ,
						intTablicaKomunikatowZnacznikZapisu := intTablicaKomunikatowZnacznikZapisu ,
						intTablicaKomunikatowRozmiar := intTablicaKomunikatowRozmiar ,
						sWyslanyKomunikat := sWyslanyKomunikatDummy);
			sDane := '';
		END_IF	
	END_IF
	//Napięcia maksymalne fazowe
	IF rMaksymalneNapiecieL1 <> rMaksymalneNapiecieL1Zaraportowana THEN
		rMaksymalneNapiecieL1Zaraportowana := rMaksymalneNapiecieL1;
		fnKomunikatDaneDodaj_xOverFlow(sDane := sDane , sAtrybut := 'VOLTMAXL1=' , sWartosc := REAL_TO_STRING(rMaksymalneNapiecieL1) , xOverFlow := xOverFlow);	
		IF xOverFlow = TRUE THEN
			fnZapiszKomunikat(	sCalyKomunikat := '' ,
						sTypKomunikatu := 'M' ,
						sMnemonik := sMnemonik ,
						sMACAdres := sMACAdres ,
						sIDNadawcy := sIdInstancji ,
						sIDOdbiorcy := sIdAplikacji ,
						sDaneZapasowe := sDaneZapasowe ,
						sDane := sDane ,
						arTablicaKomunikatow := arTablicaKomunikatow ,
						intTablicaKomunikatowZnacznikZapisu := intTablicaKomunikatowZnacznikZapisu ,
						intTablicaKomunikatowRozmiar := intTablicaKomunikatowRozmiar ,
						sWyslanyKomunikat := sWyslanyKomunikatDummy);
			sDane := '';
		END_IF	
	END_IF
	IF rMaksymalneNapiecieL2 <> rMaksymalneNapiecieL2Zaraportowana THEN
		rMaksymalneNapiecieL2Zaraportowana := rMaksymalneNapiecieL2;
		fnKomunikatDaneDodaj_xOverFlow(sDane := sDane , sAtrybut := 'VOLTMAXL2=' , sWartosc := REAL_TO_STRING(rMaksymalneNapiecieL2) , xOverFlow := xOverFlow);	
		IF xOverFlow = TRUE THEN
			fnZapiszKomunikat(	sCalyKomunikat := '' ,
						sTypKomunikatu := 'M' ,
						sMnemonik := sMnemonik ,
						sMACAdres := sMACAdres ,
						sIDNadawcy := sIdInstancji ,
						sIDOdbiorcy := sIdAplikacji ,
						sDaneZapasowe := sDaneZapasowe ,
						sDane := sDane ,
						arTablicaKomunikatow := arTablicaKomunikatow ,
						intTablicaKomunikatowZnacznikZapisu := intTablicaKomunikatowZnacznikZapisu ,
						intTablicaKomunikatowRozmiar := intTablicaKomunikatowRozmiar ,
						sWyslanyKomunikat := sWyslanyKomunikatDummy);
			sDane := '';
		END_IF	
	END_IF	
	IF rMaksymalneNapiecieL3 <> rMaksymalneNapiecieL3Zaraportowana THEN
		rMaksymalneNapiecieL3Zaraportowana := rMaksymalneNapiecieL3;
		fnKomunikatDaneDodaj_xOverFlow(sDane := sDane , sAtrybut := 'VOLTMAXL3=' , sWartosc := REAL_TO_STRING(rMaksymalneNapiecieL3) , xOverFlow := xOverFlow);	
		IF xOverFlow = TRUE THEN
			fnZapiszKomunikat(	sCalyKomunikat := '' ,
						sTypKomunikatu := 'M' ,
						sMnemonik := sMnemonik ,
						sMACAdres := sMACAdres ,
						sIDNadawcy := sIdInstancji ,
						sIDOdbiorcy := sIdAplikacji ,
						sDaneZapasowe := sDaneZapasowe ,
						sDane := sDane ,
						arTablicaKomunikatow := arTablicaKomunikatow ,
						intTablicaKomunikatowZnacznikZapisu := intTablicaKomunikatowZnacznikZapisu ,
						intTablicaKomunikatowRozmiar := intTablicaKomunikatowRozmiar ,
						sWyslanyKomunikat := sWyslanyKomunikatDummy);
			sDane := '';
		END_IF	
	END_IF
	//THD napięcia, fazowe
	IF rTHDNapieciaL1 <> rTHDNapieciaL1Zaraportowana THEN
		rTHDNapieciaL1Zaraportowana := rTHDNapieciaL1;
		fnKomunikatDaneDodaj_xOverFlow(sDane := sDane , sAtrybut := 'VOLTTHDL1=' , sWartosc := REAL_TO_STRING(rTHDNapieciaL1) , xOverFlow := xOverFlow);	
		IF xOverFlow = TRUE THEN
			fnZapiszKomunikat(	sCalyKomunikat := '' ,
						sTypKomunikatu := 'M' ,
						sMnemonik := sMnemonik ,
						sMACAdres := sMACAdres ,
						sIDNadawcy := sIdInstancji ,
						sIDOdbiorcy := sIdAplikacji ,
						sDaneZapasowe := sDaneZapasowe ,
						sDane := sDane ,
						arTablicaKomunikatow := arTablicaKomunikatow ,
						intTablicaKomunikatowZnacznikZapisu := intTablicaKomunikatowZnacznikZapisu ,
						intTablicaKomunikatowRozmiar := intTablicaKomunikatowRozmiar ,
						sWyslanyKomunikat := sWyslanyKomunikatDummy);
			sDane := '';
		END_IF	
	END_IF
	IF rTHDNapieciaL2 <> rTHDNapieciaL2Zaraportowana THEN
		rTHDNapieciaL2Zaraportowana := rTHDNapieciaL2;
		fnKomunikatDaneDodaj_xOverFlow(sDane := sDane , sAtrybut := 'VOLTTHDL2=' , sWartosc := REAL_TO_STRING(rTHDNapieciaL2) , xOverFlow := xOverFlow);	
		IF xOverFlow = TRUE THEN
			fnZapiszKomunikat(	sCalyKomunikat := '' ,
						sTypKomunikatu := 'M' ,
						sMnemonik := sMnemonik ,
						sMACAdres := sMACAdres ,
						sIDNadawcy := sIdInstancji ,
						sIDOdbiorcy := sIdAplikacji ,
						sDaneZapasowe := sDaneZapasowe ,
						sDane := sDane ,
						arTablicaKomunikatow := arTablicaKomunikatow ,
						intTablicaKomunikatowZnacznikZapisu := intTablicaKomunikatowZnacznikZapisu ,
						intTablicaKomunikatowRozmiar := intTablicaKomunikatowRozmiar ,
						sWyslanyKomunikat := sWyslanyKomunikatDummy);
			sDane := '';
		END_IF	
	END_IF
	IF rTHDNapieciaL3 <> rTHDNapieciaL3Zaraportowana THEN
		rTHDNapieciaL3Zaraportowana := rTHDNapieciaL3;
		fnKomunikatDaneDodaj_xOverFlow(sDane := sDane , sAtrybut := 'VOLTTHDL3=' , sWartosc := REAL_TO_STRING(rTHDNapieciaL3) , xOverFlow := xOverFlow);	
		IF xOverFlow = TRUE THEN
			fnZapiszKomunikat(	sCalyKomunikat := '' ,
						sTypKomunikatu := 'M' ,
						sMnemonik := sMnemonik ,
						sMACAdres := sMACAdres ,
						sIDNadawcy := sIdInstancji ,
						sIDOdbiorcy := sIdAplikacji ,
						sDaneZapasowe := sDaneZapasowe ,
						sDane := sDane ,
						arTablicaKomunikatow := arTablicaKomunikatow ,
						intTablicaKomunikatowZnacznikZapisu := intTablicaKomunikatowZnacznikZapisu ,
						intTablicaKomunikatowRozmiar := intTablicaKomunikatowRozmiar ,
						sWyslanyKomunikat := sWyslanyKomunikatDummy);
			sDane := '';
		END_IF	
	END_IF
	//THD prądu, fazowe
	IF rTHDPraduL1 <> rTHDPraduL1Zaraportowana THEN
		rTHDPraduL1Zaraportowana := rTHDPraduL1;
		fnKomunikatDaneDodaj_xOverFlow(sDane := sDane , sAtrybut := 'AMPERTHDL1=' , sWartosc := REAL_TO_STRING(rTHDPraduL1) , xOverFlow := xOverFlow);	
		IF xOverFlow = TRUE THEN
			fnZapiszKomunikat(	sCalyKomunikat := '' ,
						sTypKomunikatu := 'M' ,
						sMnemonik := sMnemonik ,
						sMACAdres := sMACAdres ,
						sIDNadawcy := sIdInstancji ,
						sIDOdbiorcy := sIdAplikacji ,
						sDaneZapasowe := sDaneZapasowe ,
						sDane := sDane ,
						arTablicaKomunikatow := arTablicaKomunikatow ,
						intTablicaKomunikatowZnacznikZapisu := intTablicaKomunikatowZnacznikZapisu ,
						intTablicaKomunikatowRozmiar := intTablicaKomunikatowRozmiar ,
						sWyslanyKomunikat := sWyslanyKomunikatDummy);
			sDane := '';
		END_IF	
	END_IF
	IF rTHDPraduL2 <> rTHDPraduL2Zaraportowana THEN
		rTHDPraduL2Zaraportowana := rTHDPraduL2;
		fnKomunikatDaneDodaj_xOverFlow(sDane := sDane , sAtrybut := 'AMPERTHDL2=' , sWartosc := REAL_TO_STRING(rTHDPraduL2) , xOverFlow := xOverFlow);
		IF xOverFlow = TRUE THEN
			fnZapiszKomunikat(	sCalyKomunikat := '' ,
						sTypKomunikatu := 'M' ,
						sMnemonik := sMnemonik ,
						sMACAdres := sMACAdres ,
						sIDNadawcy := sIdInstancji ,
						sIDOdbiorcy := sIdAplikacji ,
						sDaneZapasowe := sDaneZapasowe ,
						sDane := sDane ,
						arTablicaKomunikatow := arTablicaKomunikatow ,
						intTablicaKomunikatowZnacznikZapisu := intTablicaKomunikatowZnacznikZapisu ,
						intTablicaKomunikatowRozmiar := intTablicaKomunikatowRozmiar ,
						sWyslanyKomunikat := sWyslanyKomunikatDummy);
			sDane := '';
		END_IF		
	END_IF
	IF rTHDPraduL3 <> rTHDPraduL3Zaraportowana THEN
		rTHDPraduL3Zaraportowana := rTHDPraduL3;
		fnKomunikatDaneDodaj_xOverFlow(sDane := sDane , sAtrybut := 'AMPERTHDL3=' , sWartosc := REAL_TO_STRING(rTHDPraduL3) , xOverFlow := xOverFlow);	
		IF xOverFlow = TRUE THEN
			fnZapiszKomunikat(	sCalyKomunikat := '' ,
						sTypKomunikatu := 'M' ,
						sMnemonik := sMnemonik ,
						sMACAdres := sMACAdres ,
						sIDNadawcy := sIdInstancji ,
						sIDOdbiorcy := sIdAplikacji ,
						sDaneZapasowe := sDaneZapasowe ,
						sDane := sDane ,
						arTablicaKomunikatow := arTablicaKomunikatow ,
						intTablicaKomunikatowZnacznikZapisu := intTablicaKomunikatowZnacznikZapisu ,
						intTablicaKomunikatowRozmiar := intTablicaKomunikatowRozmiar ,
						sWyslanyKomunikat := sWyslanyKomunikatDummy);
			sDane := '';
		END_IF	
	END_IF
	IF sDane <> '' AND xPoInicjalizacji THEN
		fnZapiszKomunikat(	sCalyKomunikat := '' ,
							sTypKomunikatu := 'M' ,
							sMnemonik := sMnemonik ,
							sMACAdres := sMACAdres ,
							sIDNadawcy := sIdInstancji ,
							sIDOdbiorcy := sIdAplikacji ,
							sDaneZapasowe := sDaneZapasowe ,
							sDane := sDane ,
							arTablicaKomunikatow := arTablicaKomunikatow ,
							intTablicaKomunikatowZnacznikZapisu := intTablicaKomunikatowZnacznikZapisu ,
							intTablicaKomunikatowRozmiar := intTablicaKomunikatowRozmiar ,
							sWyslanyKomunikat := sWyslanyKomunikat);
	END_IF
END_IF

// Sprawdzanie stanu komunikacji
fbTimerBrakuKomunikacji(IN := arModbusStatusKomunikacji[bAdres] = enumModbusStatus.BrakKomunikacji, PT := T#60S);

// Sprawdzanie czy pomiar napięcia L1 działa (odczyt jest niepoprawny, jeśli nie zmienił wartości w przeciągu doby)
IF rNapiecieL1Pamiec = rNapiecieL1 THEN
	xBrakZmianyNapiecieL1 := TRUE;
ELSE
	xBrakZmianyNapiecieL1 := FALSE;	
END_IF
fbBrakZmianyNapiecieL1Timer(IN := xBrakZmianyNapiecieL1, PT := T#12H);
rNapiecieL1Pamiec := rNapiecieL1;
IF fbBrakZmianyNapiecieL1Timer.Q THEN
	xBladBrakZmianyNapiecieL1 := TRUE;
ELSE
	xBladBrakZmianyNapiecieL1 := FALSE;
END_IF

// Sprawdzanie czy pomiar napięcia L2 działa (odczyt jest niepoprawny, jeśli nie zmienił wartości w przeciągu doby)
IF rNapiecieL2Pamiec = rNapiecieL2 THEN
	xBrakZmianyNapiecieL2 := TRUE;
ELSE
	xBrakZmianyNapiecieL2 := FALSE;	
END_IF
fbBrakZmianyNapiecieL2Timer(IN := xBrakZmianyNapiecieL2, PT := T#12H);
rNapiecieL2Pamiec := rNapiecieL2;
IF fbBrakZmianyNapiecieL2Timer.Q THEN
	xBladBrakZmianyNapiecieL2 := TRUE;
ELSE
	xBladBrakZmianyNapiecieL2 := FALSE;
END_IF

// Sprawdzanie czy pomiar napięcia L3 działa (odczyt jest niepoprawny, jeśli nie zmienił wartości w przeciągu doby)
IF rNapiecieL3Pamiec = rNapiecieL3 THEN
	xBrakZmianyNapiecieL3 := TRUE;
ELSE
	xBrakZmianyNapiecieL3 := FALSE;	
END_IF
fbBrakZmianyNapiecieL3Timer(IN := xBrakZmianyNapiecieL3, PT := T#12H);
rNapiecieL3Pamiec := rNapiecieL3;
IF fbBrakZmianyNapiecieL3Timer.Q THEN
	xBladBrakZmianyNapiecieL3 := TRUE;
ELSE
	xBladBrakZmianyNapiecieL3 := FALSE;
END_IF

// Sprawdzanie czy pomiar prądu L1 działa (odczyt jest niepoprawny, jeśli nie zmienił wartości w przeciągu doby)
IF rPradL1Pamiec = rPradL1 THEN
	xBrakZmianyPradL1 := TRUE;
ELSE
	xBrakZmianyPradL1 := FALSE;	
END_IF
fbBrakZmianyPradL1Timer(IN := xBrakZmianyPradL1, PT := T#12H);
rPradL1Pamiec := rPradL1;
IF fbBrakZmianyPradL1Timer.Q THEN
	xBladBrakZmianyPradL1 := TRUE;
ELSE
	xBladBrakZmianyPradL1 := FALSE;
END_IF

// Sprawdzanie czy pomiar napięcia L2 działa (odczyt jest niepoprawny, jeśli nie zmienił wartości w przeciągu doby)
IF rPradL2Pamiec = rPradL2 THEN
	xBrakZmianyPradL2 := TRUE;
ELSE
	xBrakZmianyPradL2 := FALSE;	
END_IF
fbBrakZmianyPradL2Timer(IN := xBrakZmianyPradL2, PT := T#12H);
rPradL2Pamiec := rPradL2;
IF fbBrakZmianyPradL2Timer.Q THEN
	xBladBrakZmianyPradL2 := TRUE;
ELSE
	xBladBrakZmianyPradL2 := FALSE;
END_IF

// Sprawdzanie czy pomiar napięcia L3 działa (odczyt jest niepoprawny, jeśli nie zmienił wartości w przeciągu doby)
IF rPradL3Pamiec = rPradL3 THEN
	xBrakZmianyPradL3 := TRUE;
ELSE
	xBrakZmianyPradL3 := FALSE;	
END_IF
fbBrakZmianyPradL3Timer(IN := xBrakZmianyPradL3, PT := T#12H);
rPradL3Pamiec := rPradL3;
IF fbBrakZmianyPradL3Timer.Q THEN
	xBladBrakZmianyPradL3 := TRUE;
ELSE
	xBladBrakZmianyPradL3 := FALSE;
END_IF

// obsługa alarmów do analizatora
	//brak komunikacji z analizatorem
IF arErrorStan[enumPPPSAnalizatorDirisA40Error.BrakKomunikacji] <> enumAlarmWartosc.StanAlarmowy AND fbTimerBrakuKomunikacji.Q THEN
	arErrorStan[enumPPPSAnalizatorDirisA40Error.BrakKomunikacji] := enumAlarmWartosc.StanAlarmowy;
	arErrorKlasa[enumPPPSAnalizatorDirisA40Error.BrakKomunikacji] := enumPPPSAnalizatorDirisA40ErrorKlasa.BrakKomunikacji;
	IF xPoInicjalizacji THEN
		fnZapiszKomunikat(	sCalyKomunikat := '' ,
							sTypKomunikatu := 'E' ,
							sMnemonik := sMnemonik ,
							sMACAdres := sMACAdres ,
							sIDNadawcy := sIdInstancji ,
							sIDOdbiorcy := sIdAplikacji ,
							sDaneZapasowe := sDaneZapasowe ,
							sDane := fnKomunikatDaneError(xAktywny := TRUE , intKlasa := enumPPPSAnalizatorDirisA40ErrorKlasa.BrakKomunikacji , intNumer := enumPPPSAnalizatorDirisA40Error.BrakKomunikacji),
							arTablicaKomunikatow := arTablicaKomunikatow ,
							intTablicaKomunikatowZnacznikZapisu := intTablicaKomunikatowZnacznikZapisu ,
							intTablicaKomunikatowRozmiar := intTablicaKomunikatowRozmiar ,
							sWyslanyKomunikat := sWyslanyKomunikatDummy);
	END_IF
END_IF
IF arErrorStan[enumPPPSAnalizatorDirisA40Error.BrakKomunikacji] <> enumAlarmWartosc.StanNormalny AND NOT fbTimerBrakuKomunikacji.Q THEN
	arErrorStan[enumPPPSAnalizatorDirisA40Error.BrakKomunikacji] := enumAlarmWartosc.StanNormalny;
	arErrorKlasa[enumPPPSAnalizatorDirisA40Error.BrakKomunikacji] := enumPPPSAnalizatorDirisA40ErrorKlasa.BrakKomunikacji;
	IF xPoInicjalizacji THEN
		fnZapiszKomunikat(	sCalyKomunikat := '' ,
							sTypKomunikatu := 'E' ,
							sMnemonik := sMnemonik ,
							sMACAdres := sMACAdres ,
							sIDNadawcy := sIdInstancji ,
							sIDOdbiorcy := sIdAplikacji ,
							sDaneZapasowe := sDaneZapasowe ,
							sDane := fnKomunikatDaneError(xAktywny := FALSE , intKlasa := enumPPPSAnalizatorDirisA40ErrorKlasa.BrakKomunikacji , intNumer := enumPPPSAnalizatorDirisA40Error.BrakKomunikacji),
							arTablicaKomunikatow := arTablicaKomunikatow ,
							intTablicaKomunikatowZnacznikZapisu := intTablicaKomunikatowZnacznikZapisu ,
							intTablicaKomunikatowRozmiar := intTablicaKomunikatowRozmiar ,
							sWyslanyKomunikat := sWyslanyKomunikatDummy);
	END_IF
END_IF
	// Brak zmiany parametrów przez 24h
IF arErrorStan[enumPPPSAnalizatorDirisA40Error.BrakZmianyParametrow] <> enumAlarmWartosc.StanAlarmowy AND xBladBrakZmianyNapiecieL1 AND xBladBrakZmianyNapiecieL2 AND xBladBrakZmianyNapiecieL3 AND
   xBladBrakZmianyPradL1 AND xBladBrakZmianyPradL2 AND xBladBrakZmianyPradL3 THEN
	arErrorStan[enumPPPSAnalizatorDirisA40Error.BrakZmianyParametrow] := enumAlarmWartosc.StanAlarmowy;
	arErrorKlasa[enumPPPSAnalizatorDirisA40Error.BrakZmianyParametrow] := enumPPPSAnalizatorDirisA40ErrorKlasa.BrakZmianyParametrow;
	IF xPoInicjalizacji THEN
		fnZapiszKomunikat(	sCalyKomunikat := '' ,
							sTypKomunikatu := 'E' ,
							sMnemonik := sMnemonik ,
							sMACAdres := sMACAdres ,
							sIDNadawcy := sIdInstancji ,
							sIDOdbiorcy := sIdAplikacji ,
							sDaneZapasowe := sDaneZapasowe ,
							sDane := fnKomunikatDaneError(xAktywny := TRUE , intKlasa := enumPPPSAnalizatorDirisA40ErrorKlasa.BrakZmianyParametrow , intNumer := enumPPPSAnalizatorDirisA40Error.BrakZmianyParametrow),
							arTablicaKomunikatow := arTablicaKomunikatow ,
							intTablicaKomunikatowZnacznikZapisu := intTablicaKomunikatowZnacznikZapisu ,
							intTablicaKomunikatowRozmiar := intTablicaKomunikatowRozmiar ,
							sWyslanyKomunikat := sWyslanyKomunikatDummy);
	END_IF
END_IF
IF arErrorStan[enumPPPSAnalizatorDirisA40Error.BrakZmianyParametrow] <> enumAlarmWartosc.StanNormalny AND NOT (xBladBrakZmianyNapiecieL1 AND xBladBrakZmianyNapiecieL2 AND xBladBrakZmianyNapiecieL3 AND
   xBladBrakZmianyPradL1 AND xBladBrakZmianyPradL2 AND xBladBrakZmianyPradL3) THEN
	arErrorStan[enumPPPSAnalizatorDirisA40Error.BrakZmianyParametrow] := enumAlarmWartosc.StanNormalny;
	arErrorKlasa[enumPPPSAnalizatorDirisA40Error.BrakZmianyParametrow] := enumPPPSAnalizatorDirisA40ErrorKlasa.BrakZmianyParametrow;
	IF xPoInicjalizacji THEN
		fnZapiszKomunikat(	sCalyKomunikat := '' ,
							sTypKomunikatu := 'E' ,
							sMnemonik := sMnemonik ,
							sMACAdres := sMACAdres ,
							sIDNadawcy := sIdInstancji ,
							sIDOdbiorcy := sIdAplikacji ,
							sDaneZapasowe := sDaneZapasowe ,
							sDane := fnKomunikatDaneError(xAktywny := FALSE , intKlasa := enumPPPSAnalizatorDirisA40ErrorKlasa.BrakZmianyParametrow , intNumer := enumPPPSAnalizatorDirisA40Error.BrakZmianyParametrow),
							arTablicaKomunikatow := arTablicaKomunikatow ,
							intTablicaKomunikatowZnacznikZapisu := intTablicaKomunikatowZnacznikZapisu ,
							intTablicaKomunikatowRozmiar := intTablicaKomunikatowRozmiar ,
							sWyslanyKomunikat := sWyslanyKomunikatDummy);
	END_IF
END_IF
          
END_FUNCTION_BLOCK
